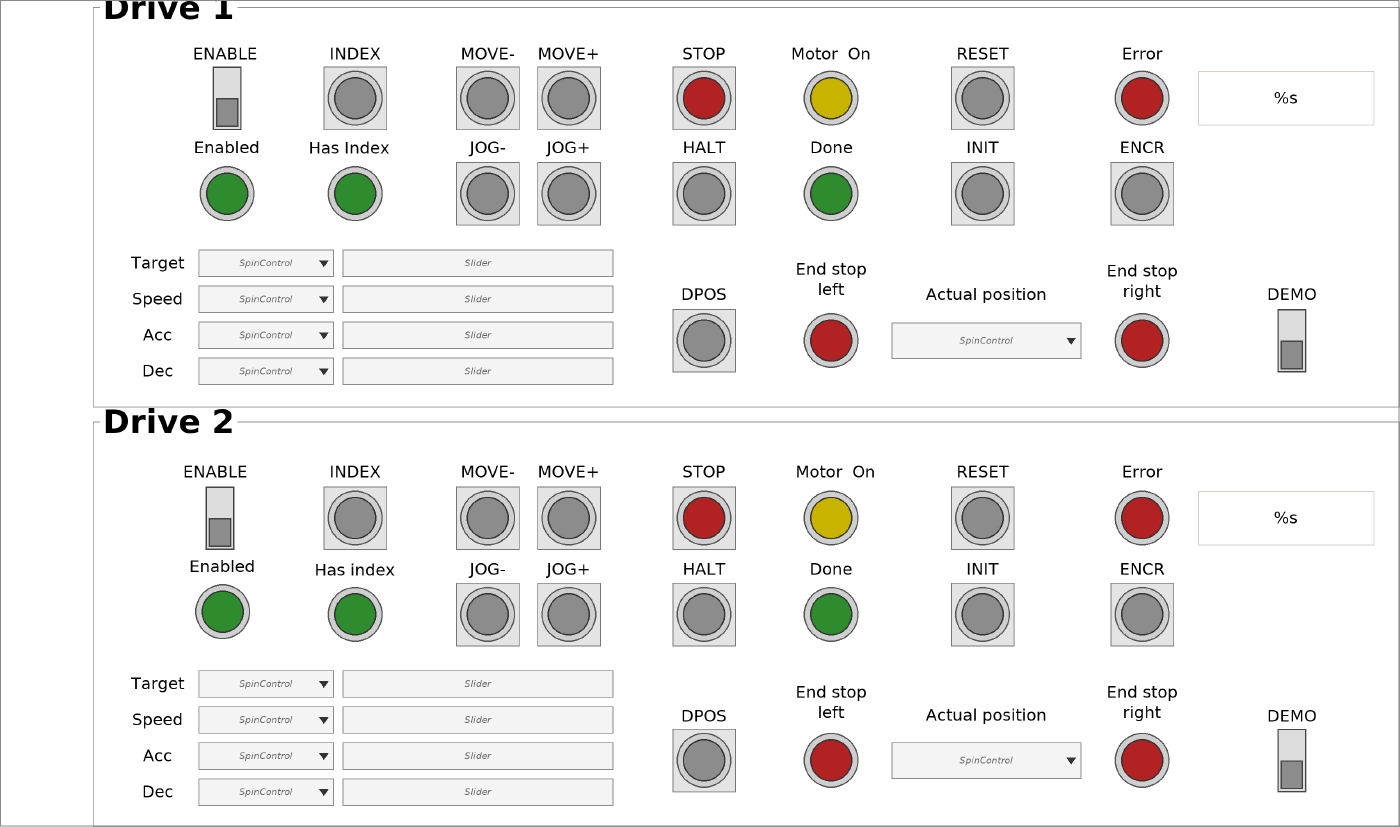
VISUALIZATION Visualization  // 1553x918
    GroupBox (103,0 1450x452), "Drive 1"
        Label (222,136 125x57), "Has Index"
        Label (762,33 114x54), "Motor On"
        PushSwitch (643,343 70x70), variable: MAIN.drive1Dpos, behaviour: TAP, style: Switch-PushSwitch-Gray
        Label (643,312 70x30), "DPOS"
        Textfield (1226,79 195x60), "%s", text variable: MAIN.drive1ErrorString
    GroupBox (103,460 1450x458), "Drive 2"
        Label (232,145 117x56), "Has index"
        Lamp1 (109,184 70x70), variable: MAIN.Drive2.iDriveAmplifiersEnabled, style: Lamp-Lamp1-Green
        Label (92,154 103x30), "Enabled"
        Label (769,38 110x52), "Motor On"
        PushSwitch (643,349 70x70), variable: MAIN.drive2Dpos, behaviour: TAP, style: Switch-PushSwitch-Gray
        Label (643,320 70x30), "DPOS"
        Label (907,319 168x30), "Actual position"
        Textfield (1226,85 195x60), "%s", text variable: MAIN.drive2ErrorString
    DipSwitch (1398,343 70x70), variable: MAIN.drive1MoveAbs, behaviour: TOGGLE, style: Switch-DipSwitch-Gray
    SpinControl (220,317 150x30), variable: MAIN.drive1Speed
    SpinControl (220,357 150x30), variable: MAIN.drive1Acc
    SpinControl (220,277 150x30), variable: MAIN.drive1Target
    SpinControl (220,397 150x30), variable: MAIN.drive1Dec
    Lamp1 (887,74 70x70), variable: MAIN.Drive1.MotorOn, style: Lamp-Lamp1-Yellow
    Lamp1 (1232,343 70x70), variable: MAIN.Drive1.RightEndstop, style: Lamp-Lamp1-Red
    Lamp1 (887,343 70x70), variable: MAIN.Drive1.LeftEndstop, style: Lamp-Lamp1-Red
    PushSwitch (1055,74 70x70), variable: MAIN.drive1Reset, behaviour: TAP, style: Switch-PushSwitch-Gray
    PushSwitch (746,74 70x70), variable: MAIN.drive1Stop, behaviour: TAP, style: Switch-PushSwitch-Red
    PushSwitch (746,180 70x70), variable: MAIN.drive1Halt, behaviour: TAP, style: Switch-PushSwitch-Gray
    PushSwitch (359,74 70x70), variable: MAIN.drive1Index, behaviour: TAP, style: Switch-PushSwitch-Gray
    Label (1388,312 90x30), "DEMO"
    Label (359,45 70x30), "INDEX"
    Label (746,149 70x30), "HALT"
    Label (746,45 70x30), "STOP"
    Label (1055,45 70x30), "RESET"
    Lamp1 (887,180 70x70), variable: MAIN.Drive1.Done, style: Lamp-Lamp1-Green
    Label (872,278 100x64), "End stop left"
    Label (1217,282 100x60), "End stop right"
    Label (877,149 91x30), "Done"
    Label (140,277 70x30), "Target"
    Label (140,317 70x30), "Speed"
    Label (140,357 70x30), "Acc"
    Label (140,397 70x30), "Dec"
    Label (1013,312 162x30), "Actual position"
    SpinControl (989,358 210x40), variable: MAIN.Drive1.ActPosition
    Slider (380,277 300x30), variable: MAIN.drive1Target, scale 0..100
    Slider (380,317 300x30), variable: MAIN.drive1Speed, scale 0..100
    Slider (380,357 300x30), variable: MAIN.drive1Acc, scale 0..100
    Slider (380,397 300x30), variable: MAIN.drive1Dec, scale 0..100
    DipSwitch (1398,809 70x70), variable: MAIN.drive2MoveAbs, behaviour: TOGGLE, style: Switch-DipSwitch-Gray
    SpinControl (220,784 150x30), variable: MAIN.drive2Speed
    SpinControl (220,824 150x30), variable: MAIN.drive2Acc
    SpinControl (220,744 150x30), variable: MAIN.drive2Target
    SpinControl (220,864 150x30), variable: MAIN.drive2Dec
    Lamp1 (887,540 70x70), variable: MAIN.Drive2.MotorOn, style: Lamp-Lamp1-Yellow
    Lamp1 (1232,809 70x70), variable: MAIN.Drive2.RightEndstop, style: Lamp-Lamp1-Red
    Lamp1 (887,809 70x70), variable: MAIN.Drive2.LeftEndstop, style: Lamp-Lamp1-Red
    PushSwitch (1055,540 70x70), variable: MAIN.drive2Reset, behaviour: TAP, style: Switch-PushSwitch-Gray
    PushSwitch (746,540 70x70), variable: MAIN.drive2Stop, behaviour: TAP, style: Switch-PushSwitch-Red
    PushSwitch (746,647 70x70), variable: MAIN.drive2Halt, behaviour: TAP, style: Switch-PushSwitch-Gray
    PushSwitch (359,540 70x70), variable: MAIN.drive2Index, behaviour: TAP, style: Switch-PushSwitch-Gray
    Label (1388,780 90x30), "DEMO"
    Label (359,509 70x30), "INDEX"
    Label (746,617 70x30), "HALT"
    Label (746,509 70x30), "STOP"
    Label (1055,509 70x30), "RESET"
    Lamp1 (887,647 70x70), variable: MAIN.Drive2.Done, style: Lamp-Lamp1-Green
    Label (872,749 100x61), "End stop left"
    Label (1217,749 100x61), "End stop right"
    Label (875,617 94x30), "Done"
    Label (140,744 70x30), "Target"
    Label (140,784 70x30), "Speed"
    Label (140,824 70x30), "Acc"
    Label (140,864 70x30), "Dec"
    SpinControl (989,824 210x40), variable: MAIN.Drive2.ActPosition
    Slider (380,744 300x30), variable: MAIN.drive2Target, scale 0..100
    Slider (380,784 300x30), variable: MAIN.drive2Speed, scale 0..100
    Slider (380,824 300x30), variable: MAIN.drive2Acc, scale 0..100
    Slider (380,864 300x30), variable: MAIN.drive2Dec, scale 0..100
    DipSwitch (217,74 70x70), variable: MAIN.drive1Enable, behaviour: TOGGLE, style: Switch-DipSwitch-Gray
    Label (200,45 100x30), "ENABLE"
    Label (189,509 100x30), "ENABLE"
    DipSwitch (209,540 70x70), variable: MAIN.drive2Enable, behaviour: TOGGLE, style: Switch-DipSwitch-Gray
    Lamp1 (359,180 70x70), variable: MAIN.Drive1.HasIndex, style: Lamp-Lamp1-Green
    Lamp1 (359,647 70x70), variable: MAIN.Drive2.HasIndex, style: Lamp-Lamp1-Green
    PushSwitch (506,180 70x70), variable: MAIN.drive1JogN, behaviour: TAP, style: Switch-PushSwitch-Gray
    PushSwitch (596,180 70x70), variable: MAIN.drive1JogP, behaviour: TAP, style: Switch-PushSwitch-Gray
    Label (506,149 70x30), "JOG-"
    Label (596,149 70x30), "JOG+"
    PushSwitch (506,647 70x70), variable: MAIN.drive2JogN, behaviour: TAP, style: Switch-PushSwitch-Gray
    PushSwitch (596,647 70x70), variable: MAIN.drive2JogP, behaviour: TAP, style: Switch-PushSwitch-Gray
    Label (506,617 70x30), "JOG-"
    Label (596,617 70x30), "JOG+"
    PushSwitch (1055,180 70x70), variable: MAIN.drive1Init, behaviour: TAP, style: Switch-PushSwitch-Gray
    Label (1055,149 70x30), "INIT"
    PushSwitch (1055,647 70x70), variable: MAIN.drive2Init, behaviour: TAP, style: Switch-PushSwitch-Gray
    Label (1055,617 70x30), "INIT"
    Lamp1 (1232,74 70x70), variable: MAIN.Drive1.HasError, style: Lamp-Lamp1-Red
    Label (1217,45 100x30), "Error"
    Lamp1 (1232,540 70x70), variable: MAIN.Drive2.HasError, style: Lamp-Lamp1-Red
    Label (1217,509 100x30), "Error"
    Lamp1 (217,180 70x70), variable: MAIN.Drive1.iDriveAmplifiersEnabled, style: Lamp-Lamp1-Green
    Label (200,149 103x30), "Enabled"
    PushSwitch (506,74 70x70), variable: MAIN.drive1MoveN, behaviour: TAP, style: Switch-PushSwitch-Gray
    PushSwitch (596,74 70x70), variable: MAIN.drive1MoveP, behaviour: TAP, style: Switch-PushSwitch-Gray
    Label (506,45 70x30), "MOVE-"
    Label (596,45 70x30), "MOVE+"
    PushSwitch (1232,180 70x70), variable: MAIN.drive1ResetEncoder, behaviour: TAP, style: Switch-PushSwitch-Gray
    Label (1223,149 88x30), "ENCR"
    PushSwitch (1232,647 70x70), variable: MAIN.drive2ResetEncoder, behaviour: TAP, style: Switch-PushSwitch-Gray
    Label (1223,617 88x30), "ENCR"
    PushSwitch (506,540 70x70), variable: MAIN.drive2MoveN, behaviour: TAP, style: Switch-PushSwitch-Gray
    PushSwitch (596,540 70x70), variable: MAIN.drive2MoveP, behaviour: TAP, style: Switch-PushSwitch-Gray
    Label (506,509 70x30), "MOVE-"
    Label (596,509 70x30), "MOVE+"
END_VISUALIZATION

(* stored: Version 1.1.0.1, ProductVersion 3.1.4024.16
   Visu Visualization: Id {4b40a633-ff4c-4025-8245-bbf0a50c9466} *)
